{attribute 'qualified_only'}
{attribute 'strict'}
{attribute 'to_string'}
TYPE ENUM_Si_B4C_Coating_States_1D :
(
     Unknown := 0,
    Si := 1,
    B4C := 2
)UINT;
END_TYPE

(* stored: Version 1.1.0.1
   DUT ENUM_Si_B4C_Coating_States_1D: Id {e4b29de5-14be-4f17-844f-a37bd25107f2} *)
